// TIA Portal V19 export
FUNCTION "FC80_TeepTrack" : Void   // FC80, LAD
{ S7_Optimized_Access := 'TRUE' }
// stored: AutoNumber false, SetENOAutomatically false
BEGIN

REGION Network 1: Teep Track Robot 1
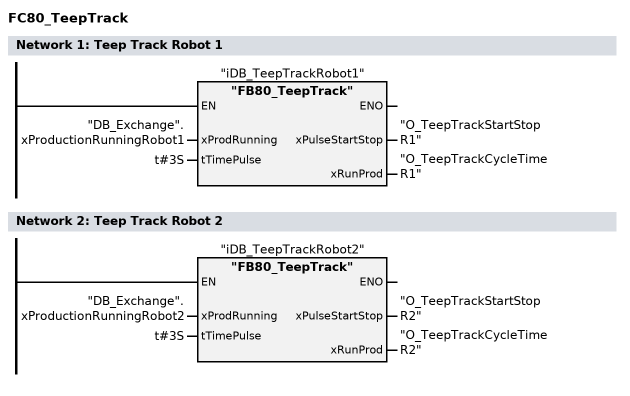
   RUNG wire#powerrail
      "iDB_TeepTrackRobot1"(xProdRunning := "DB_Exchange".xProductionRunningRobot1, tTimePulse := t#3S, xPulseStartStop => "O_TeepTrackStartStopR1", xRunProd => "O_TeepTrackCycleTimeR1")
   END_RUNG
   // the same network as SCL:
   "iDB_TeepTrackRobot1"(xProdRunning := "DB_Exchange".xProductionRunningRobot1,   // "FB80_TeepTrack"
                         tTimePulse := t#3S,
                         xPulseStartStop => "O_TeepTrackStartStopR1",
                         xRunProd => "O_TeepTrackCycleTimeR1");
END_REGION

REGION Network 2: Teep Track Robot 2
   RUNG wire#powerrail
      "iDB_TeepTrackRobot2"(xProdRunning := "DB_Exchange".xProductionRunningRobot2, tTimePulse := t#3S, xPulseStartStop => "O_TeepTrackStartStopR2", xRunProd => "O_TeepTrackCycleTimeR2")
   END_RUNG
   // the same network as SCL:
   "iDB_TeepTrackRobot2"(xProdRunning := "DB_Exchange".xProductionRunningRobot2,   // "FB80_TeepTrack"
                         tTimePulse := t#3S,
                         xPulseStartStop => "O_TeepTrackStartStopR2",
                         xRunProd => "O_TeepTrackCycleTimeR2");
END_REGION
END_FUNCTION
